FUNCTION_BLOCK SC_Dispensing (* Control of module level skill Dispensing: OPC UA Start(Session, parameters...)/Stop/Abort/Reset(Session) -> [Accepted, ErrorID]; GO starts the Execute sequence with the parameters P_*; releases its equipment at the end *)
  (* Standard: 61499-2 *)
  (* Version 0.1, 2026-09-28, Project contributors, AAU Smart Production Lab *)
  PACKAGE filling;
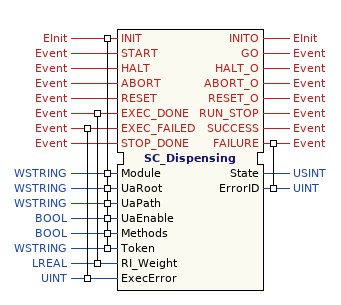
  EVENT_INPUT
    INIT : EInit WITH Module, UaRoot, UaPath, UaEnable, Methods, Token;
    START;
    HALT;
    ABORT;
    RESET;
    EXEC_DONE WITH RI_Weight;
    EXEC_FAILED WITH ExecError;
    STOP_DONE;
  END_EVENT
  EVENT_OUTPUT
    INITO : EInit;
    GO;
    HALT_O;
    ABORT_O;
    RESET_O;
    RUN_STOP;
    SUCCESS;
    FAILURE WITH ErrorID;
  END_EVENT
  VAR_INPUT
    Module : WSTRING;
    UaRoot : WSTRING;
    UaPath : WSTRING;
    UaEnable : BOOL;
    Methods : BOOL;
    Token : WSTRING;
    RI_Weight : LREAL;
    ExecError : UINT;
  END_VAR
  VAR_OUTPUT
    State : USINT;
    ErrorID : UINT;
  END_VAR
  FBS
    Control : modlib::SKILL_Control(InRange := TRUE, EqFree := TRUE);
    Params : filling::SP_Dispensing;
    Owner : modlib::MOD_OwnerView;
    Mode : modlib::MOD_StateView;
    UaStart : iec61499::net::SERVER_2_1;
    UaStop : iec61499::net::SERVER_2_1;
    UaAbort : iec61499::net::SERVER_2_1;
    UaReset : iec61499::net::SERVER_2_1;
    PubState : iec61499::net::PUBLISH_2;
    Act : iec61499::net::PUBLISH_1(QI := TRUE);
    PubResults : iec61499::net::PUBLISH_1;
    Release : modlib::SKILL_Release;
    Rel_NeedleAxis : iec61499::net::PUBLISH_4(QI := TRUE);
    Rel_Scale : iec61499::net::PUBLISH_4(QI := TRUE);
  END_FBS
  EVENT_CONNECTIONS
    Control.RSP_START TO UaStart.RSP;
    Control.RSP_STOP TO UaStop.RSP;
    Control.RSP_ABORT TO UaAbort.RSP;
    Control.RSP_RESET TO UaReset.RSP;
    UaStop.IND TO Control.CMD_STOP;
    UaAbort.IND TO Control.CMD_ABORT;
    UaReset.IND TO Control.CMD_RESET;
    UaStart.IND TO Control.CMD_START;
    Owner.CHG TO Control.OWNER_CHG;
    Mode.CHG TO Control.MOD_CHG;
    Control.PUB TO PubState.REQ;
    Control.ACT TO Act.REQ;
    START TO Control.START;
    HALT TO Control.HALT;
    ABORT TO Control.ABORT;
    RESET TO Control.RESET;
    Control.SUCCESS TO SUCCESS;
    Control.FAILURE TO FAILURE;
    INIT TO Control.INIT;
    Control.INITO TO Params.INIT;
    Params.INITO TO Owner.INIT;
    Owner.INITO TO Mode.INIT;
    Mode.INITO TO UaStart.INIT;
    UaStart.INITO TO UaStop.INIT;
    UaStop.INITO TO UaAbort.INIT;
    UaAbort.INITO TO UaReset.INIT;
    UaReset.INITO TO PubState.INIT;
    PubState.INITO TO PubResults.INIT;
    PubResults.INITO TO Act.INIT;
    Act.INITO TO Rel_NeedleAxis.INIT;
    Rel_NeedleAxis.INITO TO Rel_Scale.INIT;
    Rel_Scale.INITO TO PubState.REQ;
    Rel_Scale.INITO TO INITO;
    Control.GO_UA TO GO;
    Control.GO_PARENT TO GO;
    EXEC_DONE TO PubResults.REQ;
    EXEC_DONE TO Control.EXEC_DONE;
    EXEC_FAILED TO Control.EXEC_FAILED;
    STOP_DONE TO Control.STOP_DONE;
    Control.RUN_STOP TO RUN_STOP;
    Control.HALT_O TO HALT_O;
    Control.ABORT_O TO ABORT_O;
    Control.RESET_O TO RESET_O;
    Control.FAILURE TO Release.REQ;
    Control.ABORT_O TO Release.REQ;
    Release.CNF TO Rel_NeedleAxis.REQ;
    Release.CNF TO Rel_Scale.REQ;
  END_CONNECTIONS
  DATA_CONNECTIONS
    Module TO Control.Module;
    Module TO Owner.Module;
    Module TO Mode.Module;
    UaRoot TO Control.UaRoot;
    UaPath TO Control.UaPath;
    Module TO Params.Module;
    UaRoot TO Params.UaRoot;
    UaPath TO Params.UaPath;
    Methods TO UaStart.QI;
    Methods TO UaStop.QI;
    Methods TO UaAbort.QI;
    Methods TO UaReset.QI;
    UaEnable TO PubState.QI;
    Control.IdStart TO UaStart.ID;
    Control.Accepted TO UaStart.SD_1;
    Control.RspError TO UaStart.SD_2;
    UaStart.RD_1 TO Control.S_Start;
    Control.IdStop TO UaStop.ID;
    Control.Accepted TO UaStop.SD_1;
    Control.RspError TO UaStop.SD_2;
    UaStop.RD_1 TO Control.S_Stop;
    Control.IdAbort TO UaAbort.ID;
    Control.Accepted TO UaAbort.SD_1;
    Control.RspError TO UaAbort.SD_2;
    UaAbort.RD_1 TO Control.S_Abort;
    Control.IdReset TO UaReset.ID;
    Control.Accepted TO UaReset.SD_1;
    Control.RspError TO UaReset.SD_2;
    UaReset.RD_1 TO Control.S_Reset;
    Owner.Owner TO Control.Owner;
    Mode.State TO Control.ModState;
    Control.IdPub TO PubState.ID;
    Control.State TO PubState.SD_1;
    Control.State TO State;
    Control.ErrorID TO PubState.SD_2;
    Control.ErrorID TO ErrorID;
    Control.IdAct TO Act.ID;
    Control.Delta TO Act.SD_1;
    UaEnable TO PubResults.QI;
    Params.IdResults TO PubResults.ID;
    RI_Weight TO PubResults.SD_1;
    ExecError TO Control.ExecError;
    Token TO Release.Token;
    Params.IdRel_NeedleAxis TO Rel_NeedleAxis.ID;
    Release.Holder TO Rel_NeedleAxis.SD_1;
    Release.Command TO Rel_NeedleAxis.SD_2;
    Release.Arg TO Rel_NeedleAxis.SD_3;
    Release.Release TO Rel_NeedleAxis.SD_4;
    Params.IdRel_Scale TO Rel_Scale.ID;
    Release.Holder TO Rel_Scale.SD_1;
    Release.Command TO Rel_Scale.SD_2;
    Release.Arg TO Rel_Scale.SD_3;
    Release.Release TO Rel_Scale.SD_4;
  END_CONNECTIONS
END_FUNCTION_BLOCK
